{attribute 'GeneratedUsingTerminal: IODEVICETYPE_ETHERCATPROT'}
{attribute addProperty BoxType "IODEVICETYPE_ETHERCATPROT"}
{attribute addProperty Id "boxesboxes_1045F1DB5785A_0076_AMP8000_0030_0103AMP8000_7C531350113SyncUnitsSyncUnits_99E584AF18InputsInputs_25A0042B160OutputsOutputs_2397A10E106InfoDataInfoData_E68C61CD28"}
{attribute addProperty CRC "4288671729"}
{attribute addProperty Size "6210"}
TYPE EtherCAT_Master_Duplicates_FF9FEFF1 :
STRUCT
	{attribute addProperty Name "boxes"}
	boxes : boxes_1045F1DB;
	{attribute addProperty Name "A_0076_AMP8000_0030_0103"}
	A_0076_AMP8000_0030_0103 : AMP8000_7C531350;
	{attribute addProperty Name "SyncUnits"}
	SyncUnits : SyncUnits_99E584AF;
	{attribute addProperty Name "Inputs"}
	Inputs : Inputs_25A0042B;
	{attribute addProperty Name "Outputs"}
	Outputs : Outputs_2397A10E;
	{attribute addProperty Name "InfoData"}
	InfoData : InfoData_E68C61CD;
END_STRUCT
END_TYPE

(* stored: Version 1.2.0.0, ProductVersion 3.1.4024.9
   DUT EtherCAT_Master_Duplicates_FF9FEFF1: Id {69a1f170-d932-4377-b393-c3bc2cdf0302} *)
